# EPICS StreamDevice protocol: tlPM100App/Db/tlPM100.proto
#
# Example prototype entries for USB TMC (488) devices
#

#
# Disconnect (and likely auto-reconnect) whenever anything goes wrong.
#
@mismatch     { disconnect; }
@writetimeout { disconnect; }
@readtimeout  { disconnect; }
@replyTimeout { disconnect; }

#
# Get a string value, size is passed as second argument
#
getString {
    out "\$1?";
    in "%\$2[^\r\n]";
    ExtraInput = Ignore;
}

#
# Send a command
#
cmd {
    out "\$1";
}

#
# Get an integer (decimal) value
#
getD {
    out "\$1?";
    in "%d";
    ExtraInput = Ignore;
}

#
# Set an integer (decimal) value
# Read back initial value on startup
#
setD {
    @init { out "\$1?"; in "%d"; }
    out "\$1 %d";
    ExtraInput = Ignore;
}

#
# Get a floating-point value
#
getF {
    out "\$1?";
    in "%f";
    ExtraInput = Ignore;
}

#
# Set a floating-point value
# Read back initial value on startup
#
setF {
    @init { out "\$1?"; in "%f"; }
    out "\$1 %f";
    ExtraInput = Ignore;
}

setString {
#    @init { out "\$1?"; in "%f"; }
    out "\$1 %s";
    ExtraInput = Ignore;
}
